# EPICS autosave request: iocBoot/sioc-esb-lsc01/lsc.req
$(P):IOC.DESC
$(P):FREERUN:NCYCLES
$(P):DELAY:MIN
$(P):DELAY:SEC
$(P):DELAY:MSEC
$(P):EXPOSURE:MIN
$(P):EXPOSURE:SEC
$(P):EXPOSURE:MSEC
